(* IEC 61131-3 sources: POMIRTS_lab3/AS/Library/AsMbTCP, 3 files *)

(* ---- AsMbTCP.typ ---- *)
(********************************************************************
 * COPYRIGHT -- Bernecker + Rainer
 ********************************************************************
 * Library: AsMbTCP
 * File: AsMbTCP.typ
 * Author: B+R
 ********************************************************************
 * Data types of library AsMbTCP
 ********************************************************************)

TYPE

END_TYPE

(* ---- AsMbTCP.fun ---- *)
(********************************************************************
 * COPYRIGHT -- Bernecker + Rainer
 ********************************************************************
 * Library: AsMbTCP
 * File: AsMbTCP.fun
 * Author: B+R
 ********************************************************************
 * Functions and function blocks of library AsMbTCP
 ********************************************************************)

FUNCTION_BLOCK mbReadCoils							(*mfc Read Coils; asynchronous execution*)
	VAR_INPUT
		enable			: BOOL;						(*enables execution*)
		pStation		: UDINT;					(*pointer to the station path e.g."IF2.ST1"*)
		startAddress	: UINT;						(*starting address*)
		nrCoils			: UINT;						(*number of coils to read*)
		pData			: UDINT;					(*pointer to local storage*)
		dataSize		: UINT;						(*size of local storage*)
	END_VAR

	VAR
		i_buffer		: ARRAY[0..249] OF USINT;	(*internal variable*)
        i_queryID		: UDINT;					(*internal variable*)
		i_hInstance		: UDINT;					(*internal variable*)
		i_hMbCons		: UDINT;					(*internal variable*)
		i_state			: UINT;						(*internal variable*)
	END_VAR

	VAR_OUTPUT
		status			: UINT;						(*execution status: ERR_OK, ERR_FUB_ENABLE_FALSE, ERR_FUB_BUSY, 0xXXXX = see help*)
	END_VAR
END_FUNCTION_BLOCK

FUNCTION_BLOCK mbReadDiscreteInputs					(*mfc Read Discrete Inputs; asynchronous execution*)
	VAR_INPUT
		enable			: BOOL;						(*enables execution*)
		pStation		: UDINT;					(*pointer to the station path e.g."IF2.ST1"*)
		startAddress	: UINT;						(*starting address*)
		nrInputs		: UINT;						(*number of inputs to read*)
		pData			: UDINT;					(*pointer to local storage*)
		dataSize		: UINT;						(*size of local storage*)
	END_VAR

	VAR
		i_buffer		: ARRAY[0..249] OF USINT;	(*internal variable*)
        i_queryID		: UDINT;					(*internal variable*)
		i_hInstance		: UDINT;					(*internal variable*)
		i_hMbCons		: UDINT;					(*internal variable*)
		i_state			: UINT;						(*internal variable*)
	END_VAR

	VAR_OUTPUT
		status			: UINT;						(*execution status: ERR_OK, ERR_FUB_ENABLE_FALSE, ERR_FUB_BUSY, 0xXXXX = see help*)
	END_VAR
END_FUNCTION_BLOCK

FUNCTION_BLOCK mbReadHoldingRegisters		(*mfc Read Holding Registers; asynchronous execution*)
	VAR_INPUT
		enable			: BOOL;				(*enables execution*)
		pStation		: UDINT;			(*pointer to the station path e.g. "IF2.ST1"*)
		startAddress	: UINT;				(*starting address*)
		nrRegisters		: UINT;				(*number of holding registers to read*)
		pData			: UDINT;			(*pointer to local storage*)
		dataSize		: UINT;				(*size of local storage*)
	END_VAR

	VAR
        i_queryID		: UDINT;			(*internal variable*)
		i_hInstance		: UDINT;			(*internal variable*)
		i_hMbCons		: UDINT;			(*internal variable*)
		i_state			: UINT;				(*internal variable*)
	END_VAR

	VAR_OUTPUT
		status			: UINT;				(*execution status: ERR_OK, ERR_FUB_ENABLE_FALSE, ERR_FUB_BUSY, 0xXXXX = see help*)
	END_VAR
END_FUNCTION_BLOCK

FUNCTION_BLOCK mbReadInputRegisters			(*mfc Read Input Register; asynchronous execution*)
	VAR_INPUT
		enable			: BOOL;				(*enables execution*)
		pStation		: UDINT;			(*pointer to the station path e.g."IF2.ST1"*)
		startAddress	: UINT;				(*starting address*)
		nrRegisters		: UINT;				(*number of registers to read*)
		pData			: UDINT;			(*pointer to local storage*)
		dataSize		: UINT;				(*size of local storage*)
	END_VAR

	VAR
        i_queryID		: UDINT;			(*internal variable*)
		i_hInstance		: UDINT;			(*internal variable*)
		i_hMbCons		: UDINT;			(*internal variable*)
		i_state			: UINT;				(*internal variable*)
	END_VAR

	VAR_OUTPUT
		status			: UINT;				(*execution status: ERR_OK, ERR_FUB_ENABLE_FALSE, ERR_FUB_BUSY, 0xXXXX = see help*)
	END_VAR
END_FUNCTION_BLOCK

FUNCTION_BLOCK mbWriteSingleCoil			(*mfc Write Single Coil; asynchronous execution*)
	VAR_INPUT
		enable			: BOOL;				(*enables execution*)
		pStation		: UDINT;			(*pointer to the station path e.g."IF2.ST1"*)
		startAddress	: UINT;				(*starting address*)
		value			: BOOL;				(*value to write*)
	END_VAR

	VAR
        i_queryID		: UDINT;			(*internal variable*)
		i_hInstance		: UDINT;			(*internal variable*)
		i_hMbCons		: UDINT;			(*internal variable*)
		i_state			: UINT;				(*internal variable*)
	END_VAR

	VAR_OUTPUT
		status			: UINT;				(*execution status: ERR_OK, ERR_FUB_ENABLE_FALSE, ERR_FUB_BUSY, 0xXXXX = see help*)
	END_VAR
END_FUNCTION_BLOCK

FUNCTION_BLOCK mbWriteSingleRegister		(*mfc Write Single Register; asynchronous execution*)
	VAR_INPUT
		enable			: BOOL;				(*enables execution*)
		pStation		: UDINT;			(*pointer to the station path e.g."IF2.ST1"*)
		startAddress	: UINT;				(*starting address*)
		value			: UINT;				(*value to write*)
	END_VAR

	VAR
        i_queryID		: UDINT;			(*internal variable*)
		i_hInstance		: UDINT;			(*internal variable*)
		i_hMbCons		: UDINT;			(*internal variable*)
		i_state			: UINT;				(*internal variable*)
	END_VAR

	VAR_OUTPUT
		status			: UINT;				(*execution status: ERR_OK, ERR_FUB_ENABLE_FALSE, ERR_FUB_BUSY, 0xXXXX = see help*)
	END_VAR
END_FUNCTION_BLOCK

FUNCTION_BLOCK mbWriteMultipleCoils					(*mfc Write Multiple Coils; asynchronous execution*)
	VAR_INPUT
		enable			: BOOL;						(*enables execution*)
		pStation		: UDINT;					(*pointer to the station path e.g."IF2.ST1"*)
		startAddress	: UINT;						(*starting address*)
		nrCoils			: UINT;						(*number of coils to write*)
		pData			: UDINT;					(*pointer to local storage*)
		dataSize		: UINT;						(*size of local storage*)
	END_VAR

	VAR
		i_buffer		: ARRAY[0..249] OF USINT;	(*internal variable*)
        i_queryID		: UDINT;					(*internal variable*)
		i_hInstance		: UDINT;					(*internal variable*)
		i_hMbCons		: UDINT;					(*internal variable*)
		i_state			: UINT;						(*internal variable*)
	END_VAR

	VAR_OUTPUT
		status			: UINT;						(*execution status: ERR_OK, ERR_FUB_ENABLE_FALSE, ERR_FUB_BUSY, 0xXXXX = see help*)
	END_VAR
END_FUNCTION_BLOCK

FUNCTION_BLOCK mbWriteMultipleRegisters		(*mfc Write Multiple Registers; asynchronous execution*)
	VAR_INPUT
		enable			: BOOL;				(*enables execution*)
		pStation		: UDINT;			(*pointer to the station path e.g."IF2.ST1"*)
		startAddress	: UINT;				(*starting address*)
		nrRegisters		: UINT;				(*number of registers to write*)
		pData			: UDINT;			(*pointer to local storage*)
		dataSize		: UINT;				(*size of local storage*)
	END_VAR

	VAR
        i_queryID		: UDINT;			(*internal variable*)
		i_hInstance		: UDINT;			(*internal variable*)
		i_hMbCons		: UDINT;			(*internal variable*)
		i_state			: UINT;				(*internal variable*)
	END_VAR

	VAR_OUTPUT
		status			: UINT;				(*execution status: ERR_OK, ERR_FUB_ENABLE_FALSE, ERR_FUB_BUSY, 0xXXXX = see help*)
	END_VAR
END_FUNCTION_BLOCK

FUNCTION_BLOCK mbReadWriteMultipleRegisters	(*mfc Read Write Multiple Registers; asynchronous execution*)
	VAR_INPUT
		enable				: BOOL;			(*enables execution*)
		pStation			: UDINT;		(*pointer to the station path e.g."IF2.ST1"*)
		startAddressRead	: UINT;			(*starting address for read*)
		nrRegistersRead		: UINT;			(*number of registers to read*)
		pDataRead			: UDINT;		(*pointer to local storage for read data*)
		dataSizeRead		: UINT;			(*size of local storage for read data*)
		startAddressWrite	: UINT;			(*starting address for write*)
		nrRegistersWrite	: UINT;			(*number of registers to write*)
		pDataWrite			: UDINT;		(*pointer to local storage for write data*)
		dataSizeWrite		: UINT;			(*size of local storage for write data*)
	END_VAR

	VAR
        i_queryID		: UDINT;			(*internal variable*)
		i_hInstance		: UDINT;			(*internal variable*)
		i_hMbCons		: UDINT;			(*internal variable*)
		i_state			: UINT;				(*internal variable*)
	END_VAR

	VAR_OUTPUT
		status			: UINT;				(*execution status: ERR_OK, ERR_FUB_ENABLE_FALSE, ERR_FUB_BUSY, 0xXXXX = see help*)
	END_VAR
END_FUNCTION_BLOCK

FUNCTION_BLOCK mbGetLastException			(*get last modbus exception; asynchronous execution*)
	VAR_INPUT
		enable				: BOOL;			(*enables execution*)
		pStation			: UDINT;		(*pointer to the station path e.g."IF2.ST1"*)
	END_VAR

	VAR_OUTPUT
		mbExcp				: USINT;		(*last modbus exception*)
		status				: UINT;			(*execution status: ERR_OK, ERR_FUB_ENABLE_FALSE, ERR_FUB_BUSY, 0xXXXX = see help*)
	END_VAR
END_FUNCTION_BLOCK

(* ---- AsMbTCP.var ---- *)
(********************************************************************
 * COPYRIGHT -- Bernecker + Rainer
 ********************************************************************
 * Library: AsMbTCP
 * File: AsMbTCP.var
 * Author: B+R
 ********************************************************************
 * Local variables of library AsMbTCP
 ********************************************************************)

VAR CONSTANT

	mbERR_STATION_NOT_EXIST				: UDINT := 34200;		(*station does not exist*)
	mbERR_STATION_NOT_CONNECTED			: UDINT := 34201;		(*station is not connected*)
	mbERR_INVALID_NUMBER				: UDINT := 34202;		(*number of coils/registers incorrect*)
	mbERR_NULLPOINTER					: UDINT := 34203;		(*nullpointer*)
	mbERR_DATASIZE						: UDINT := 34204;		(*storage is too small*)
	mbERR_EXCEPTION						: UDINT := 34205;		(*modbus response contains an exception*)
	mbERR_REFRESH_TIME_VIOLATION		: UDINT := 34206;		(*refresh time violation*)
	mbERR_QUEUE_OVL						: UDINT := 34207;		(*queue overload*)

	mbMFC_READ_COILS					: UDINT	:= 1;			(*mfc read coils*)
	mbMFC_READ_DISCRETE_INPUTS			: UDINT	:= 2;			(*mfc read discrete inputs*)
	mbMFC_READ_HOLDING_REGISTERS		: UDINT	:= 3;			(*mfc read holding registers*)
	mbMFC_READ_INPUT_REGISTERS			: UDINT	:= 4;			(*mfc read input register*)
	mbMFC_WRITE_SINGLE_COIL				: UDINT	:= 5;			(*mfc write single coil*)
	mbMFC_WRITE_SINGLE_REGISTER			: UDINT	:= 6;			(*mfc write single register*)
	mbMFC_WRITE_MULTIPLE_COILS			: UDINT	:= 15;			(*mfc write multiple coils*)
	mbMFC_WRITE_MULTIPLE_REGISTERS		: UDINT	:= 16;			(*mfc write multiple registers*)
	mbMFC_READ_WRITE_MULTIPLE_REG		: UDINT	:= 23;			(*mfc read write multiple registers*)
END_VAR
